FUNCTION_BLOCK FB_Conveyor EXTENDS FB_Peer IMPLEMENTS I_Module
VAR_INPUT
	in_bSystemStart : BOOL;
	in_bStop : BOOL;
	in_bStart : BOOL;
END_VAR
VAR_OUTPUT
	out_fbSensorStop : FB_Sensor;
	out_fbSensorMaterialDispatch : FB_Sensor;
	out_fbSensorSignal : FB_Sensor;
END_VAR
VAR	
	{attribute 'OPC.UA.DA' := '1'}
	bStartMotor AT%Q* : BOOL;
	iSequence : I_ConveyorSequence;
	sModuleName : STRING;
END_VAR

M_CallComponents();
IF in_bSystemStart THEN
	M_RunSequence();
END_IF

PROPERTY AccessModuleName : STRING
GET
AccessModuleName := sModuleName;
END_GET
SET
sModuleName := AccessModuleName;
END_SET
END_PROPERTY

METHOD M_CallComponents : E_PeerReturnCode
VAR_INPUT
END_VAR
out_fbSensorSignal();
out_fbSensorMaterialDispatch();
out_fbSensorStop();
END_METHOD

METHOD M_RegisterSequence : BOOL
VAR_INPUT
	in_iSequence : I_ConveyorSequence;
END_VAR
iSequence := in_iSequence;
END_METHOD

METHOD M_RunSequence : BOOL
VAR_INPUT
END_VAR
IF iSequence = NULL THEN
	RETURN;
END_IF

iSequence.M_ConveyorSequence(this^);
END_METHOD

METHOD M_StartConveyor : BOOL
VAR_INPUT
END_VAR
bStartMotor := TRUE;
END_METHOD

METHOD M_StopConveyor : E_PeerReturnCode
VAR_INPUT
END_VAR
bStartMotor := FALSE;
END_METHOD

END_FUNCTION_BLOCK

(* stored: Version 1.1.0.1, ProductVersion 3.1.4022.16
   POU FB_Conveyor: Id {69450c1a-ee4c-47aa-99f8-d851169b590d}, SpecialFunc None
   Property AccessModuleName: Id {5f009d0a-4ed1-4a9b-be38-06234da4c685}
   Get Get: Id {4de1b51f-a881-46e7-aeaf-b75ed26efacb}
   Set Set: Id {0aa9c80f-ba61-4613-8c1c-00e862dd5304}
   Method M_CallComponents: Id {d771bb4b-f7bb-488a-9824-3c6594412706}
   Method M_RegisterSequence: Id {1da2d62e-6caa-40e2-94d1-af7e92fd682d}
   Method M_RunSequence: Id {338a3dfd-c235-4a82-9dba-a5051aee481c}
   Method M_StartConveyor: Id {63eaa96e-8dac-4661-a1f7-5f07796fa619}
   Method M_StopConveyor: Id {a0f92c9a-6afa-476a-ab86-88f9d155234b} *)
